# EPICS substitutions: iocs/B22OpticsBox/B22OpticsBoxApp/Db/B22OpticsBox_expanded.substitutions
# This file was automatically generated on Fri 03 Aug 2012 11:51:40 BST from
# source: /dls_sw/prod/R3.14.11/support/pmacCoord/1-11/etc/makeIocs/B22OpticsBox.xml
#
# *** Please do not edit this file: edit the source file instead. ***
#

# Macros:
#  P           Device Prefix
#  M           Device Suffix
#  PORT        Asyn port for motor record
#  ADDR        Address on controller
#  DESC        Description, displayed on EDM screen
#  MRES        Motor Step Size (EGU)
#  VELO        Velocity (EGU/s)
#  PREC        Display Precision
#  EGU         Engineering Units
#  DHLM        Dial High Limit
#  DLLM        Dial Low Limit
#  TWV         Tweak Step Size (EGU)
#  DTYP        DTYP of record
#  DIR         User Direction
#  VBAS        Base Velocity (EGU/s)
#  VMAX        Max Velocity (EGU/s), defaults to VELO
#  ACCL        Seconds to Velocity
#  BDST        BL Distance (EGU)
#  BVEL        BL Velocity (EGU/s)
#  BACC        BL Seconds to Veloc.
#  HLSV        HW Lim. Violation Svr
#  INIT        Startup commands
#  SREV        Steps per Revolution
#  RRES        Readback Step Size (EGU)
#  ERES        Encoder Step Size (EGU)
#  JAR         Jog Acceleration (EGU/s^2)
#  UEIP        Use Encoder If Present
#  URIP        Use RDBL If Present
#  RDBL        Readback Location, set URIP = 1 if you specify this
#  RTRY        Max retry count
#  DLY         Readback settle time (s)
#  OFF         User Offset (EGU)
#  RDBD        Retry Deadband (EGU)
#  FOFF        Freeze Offset, 0=variable, 1=frozen
#  ADEL        Alarm monitor deadband (EGU)
#  NTM         New Target Monitor, only set to 0 for soft motors
#  FEHIGH      HIGH limit for following error
#  FEHIHI      HIHI limit for following error
#  FEHHSV      HIHI alarm severity for following error
#  FEHSV       HIGH alarm severity for following error
#  SCALE       Scale factor, if pmacSetAxisScale is used this should be set
#  HOMEVIS     If 1 then home is visible on the gui
#  HOMEVISSTR  If HOMEVIS=0, then display this text on the gui instead
#  name        Object name and gui association name
#  alh         Set this to alh to add the motor to the alarm handler and send emails,
#  gda_name    Name to export this as to GDA
#  gda_desc    Description to export this as to GDA
file $(MOTOR)/db/basic_asyn_motor.template
{
pattern { P, M, PORT, ADDR, DESC, MRES, VELO, PREC, EGU, DHLM, DLLM, TWV, DTYP, DIR, VBAS, VMAX, ACCL, BDST, BVEL, BACC, HLSV, INIT, SREV, RRES, ERES, JAR, UEIP, URIP, RDBL, RTRY, DLY, OFF, RDBD, FOFF, ADEL, NTM, FEHIGH, FEHIHI, FEHHSV, FEHSV, SCALE, HOMEVIS, HOMEVISSTR, name, alh, gda_name, gda_desc }
    { "B22OPTICSBOX", ":M9P", "BRICK1", "1", "M9 Pitch", "0.001", "1", "3", "mm", "1000", "-1000", "0.1", "asynMotor", "0", "0", "$(VELO)", "0.5", "0", "0", "", "MAJOR", "", "1000", "", "", "", "0", "0", "", "0", "0", "2", "", "0", "0", "1", "0", "0", "NO_ALARM", "NO_ALARM", "1", "1", "Use motor summary screen", "BOX1.M9P", "None", "", "$(DESC)" }
    { "B22OPTICSBOX", ":M9R", "BRICK1", "2", "M9 Roll", "0.001", "1", "3", "mm", "1000", "-1000", "0.1", "asynMotor", "0", "0", "$(VELO)", "0.5", "0", "0", "", "MAJOR", "", "1000", "", "", "", "0", "0", "", "0", "0", "3", "", "0", "0", "1", "0", "0", "NO_ALARM", "NO_ALARM", "1", "1", "Use motor summary screen", "BOX1.M9R", "None", "", "$(DESC)" }
    { "B22OPTICSBOX", ":M10P", "BRICK1", "3", "M10 Pitch", "0.001", "1", "3", "mm", "1000", "-1000", "0.1", "asynMotor", "0", "0", "$(VELO)", "0.5", "0", "0", "", "MAJOR", "", "1000", "", "", "", "0", "0", "", "0", "0", "4", "", "0", "0", "1", "0", "0", "NO_ALARM", "NO_ALARM", "1", "1", "Use motor summary screen", "BOX1.M10P", "None", "", "$(DESC)" }
    { "B22OPTICSBOX", ":M10R", "BRICK1", "4", "M10 Roll", "0.001", "1", "3", "mm", "1000", "-1000", "0.1", "asynMotor", "0", "0", "$(VELO)", "0.5", "0", "0", "", "MAJOR", "", "1000", "", "", "", "0", "0", "", "0", "0", "0", "", "0", "0", "1", "0", "0", "NO_ALARM", "NO_ALARM", "1", "1", "Use motor summary screen", "BOX1.M10R", "None", "", "$(DESC)" }
    { "B22OPTICSBOX", ":XEXIT", "BRICK1CS2", "5", "X Exit (compound)", "0.0001", "1", "3", "mm", "1000", "-1000", "0.1", "asynMotor", "0", "0", "$(VELO)", "0.5", "0", "0", "", "MAJOR", "", "1000", "", "", "", "0", "0", "", "0", "0", "0", "", "0", "0", "1", "0", "0", "NO_ALARM", "NO_ALARM", "1", "1", "Use motor summary screen", "BOX1.XEXIT", "None", "", "$(DESC)" }
    { "B22OPTICSBOX", ":YEXIT", "BRICK1CS2", "6", "Y Exit (compound)", "0.0001", "1", "3", "mm", "1000", "-1000", "0.1", "asynMotor", "0", "0", "$(VELO)", "0.5", "0", "0", "", "MAJOR", "", "1000", "", "", "", "0", "0", "", "0", "0", "0", "", "0", "0", "1", "0", "0", "NO_ALARM", "NO_ALARM", "1", "1", "Use motor summary screen", "BOX1.YEXIT", "None", "", "$(DESC)" }
    { "B22OPTICSBOX", ":THETAEXIT", "BRICK1CS2", "7", "Theta Exit (compound)", "0.0001", "1", "3", "rad", "1000", "-1000", "0.1", "asynMotor", "0", "0", "$(VELO)", "0.5", "0", "0", "", "MAJOR", "", "1000", "", "", "", "0", "0", "", "0", "0", "0", "", "0", "0", "1", "0", "0", "NO_ALARM", "NO_ALARM", "1", "1", "Use motor summary screen", "BOX1.THETAEXIT", "None", "", "$(DESC)" }
    { "B22OPTICSBOX", ":PHIEXIT", "BRICK1CS2", "8", "Phi Exit (compound)", "0.0001", "1", "3", "rad", "1000", "-1000", "0.1", "asynMotor", "0", "0", "$(VELO)", "0.5", "0", "0", "", "MAJOR", "", "1000", "", "", "", "0", "0", "", "0", "0", "0", "", "0", "0", "1", "0", "0", "NO_ALARM", "NO_ALARM", "1", "1", "Use motor summary screen", "BOX1.PHIEXIT", "None", "", "$(DESC)" }
}

# Macros:
#  P      Template argument
#  M      Template argument
#  SPORT  Template argument
file $(PMACCOORD)/db/motor_in_cs.template
{
pattern { P, M, SPORT }
    { "B22OPTICSBOX", ":M9P", "BRICK1port" }
    { "B22OPTICSBOX", ":M9R", "BRICK1port" }
    { "B22OPTICSBOX", ":M10P", "BRICK1port" }
    { "B22OPTICSBOX", ":M10R", "BRICK1port" }
}

# Macros:
#  P      Pv Prefix
#  PORT   Delta tau motor controller comms port
#  COORD  Co-ordinate system number
#  PREC   Precision to display variables
#  name   Object name and gui association name
file $(PMACCOORD)/db/B22_optics_box.template
{
pattern { P, PORT, COORD, PREC, name }
    { "B22OPTICSBOX", "BRICK1port", "2", "3", "BOX1.SETUP" }
}
